PROGRAM MAIN
VAR
	
	httpClient : FB_IotHttpClient :=(sHostName:='postman-echo.com',bKeepAlive:=TRUE ,tConnectionTimeout:=T#10S);
	
	request			: FB_IotHttpRequest;
	trigger : BOOL ;
	state : (INIT, SEND_REQUEST, WAIT_FOR_RESPONS, READ_RESPONSE, ERROR);
	debugRequestContent : STRING(511);
	jsonParser : FB_JsonDomParser;
	jsonDocument : SJsonValue;
	jsonArgsMember : SJsonValue;
	jsonFoo2Member : SJsonValue;
	result : STRING ; 
	isBusy : BOOL;
	
END_VAR

//init client parameters at startup
IF NOT httpClient.bConfigured THEN
httpClient.nHostPort:= 443; // Default 80
//httpClient.stTLS.bNoServerCertCheck:= TRUE;
END_IF

IF httpClient.bConfigured THEN
	
	CASE state OF
		
	INIT:
	
		IF trigger THEN
			
			state :=  SEND_REQUEST;	
			trigger := FALSE;
			
		END_IF
	
	SEND_REQUEST:
	
		IF request.SendRequest(sUri:='/get?foo1=bar1&foo2=bar2', fbClient:=httpClient, eRequestType:=ETcIotHttpRequestType.HTTP_Get, 0, 0, 0) THEN
			
			isBusy := request.bBusy;				
			state := WAIT_FOR_RESPONS;
			
		END_IF
	WAIT_FOR_RESPONS:
		
		IF request.bError THEN
			state := ERROR;
		END_IF
	
		IF NOT request.bBusy THEN // remove NOT to test 																																																																																																																	
			state :=  READ_RESPONSE;
		END_IF
		
		
	READ_RESPONSE:
	
		request.GetContent(pContent:= ADR(debugRequestContent), nContentSize:= SIZEOF(debugRequestContent), bSetNullTermination:= TRUE);
		IF request.nStatusCode >= 200 AND request.nStatusCode < 300 THEN
			jsonDocument:= request.GetJsonDomContent(jsonParser);
			IF jsonDocument <> 0 THEN
				IF jsonParser.HasMember(jsonDocument, 'args')  THEN
					jsonArgsMember:= jsonParser.FindMember(jsonDocument, 'args');
					IF jsonParser.HasMember(jsonArgsMember, 'foo2')  THEN
						jsonFoo2Member:= jsonParser.FindMember(jsonArgsMember, 'foo2');
								 					
						IF jsonParser.IsString(jsonFoo2Member) THEN							
							result:= jsonParser.GetString(jsonFoo2Member);									
						END_IF
					END_IF
					
				END_IF
				
			END_IF
					
		END_IF
		state:= INIT;
		
	ERROR:
		//
		
	END_CASE
END_IF

httpClient.Execute();

END_PROGRAM

(* stored: Version 1.1.0.1, ProductVersion 3.1.4024.13
   POU MAIN: Id {69930fcc-4ccd-4371-8944-33e8c0b2d73b}, SpecialFunc None *)
